(*
Nazwa:			GVL_VIS
Opis:			Zmienne dla wizualizacji
Wersja:			v0.2
Data:			2024-02-20
Autor:			MK
Urzadzenia:		
Konfiguracja:	
Info:
Zmiany:
- 20240220 [DP] Poprawki przed nowa wizką
*)

{attribute 'qualified_only'}
VAR_GLOBAL
	(*Legenda dla wizki :
		[H] - Hidden, prawdopodobnie nie potrzebne
		[I] - Info, informacja,
		[L] - Later, do zrobienia później, być może do przerobienia
	Uprawienia:
		brak opisu - operator
		[m] - Meechanik i powyżej
		[t] - Technolog i powyżej
		[s] - Serwis i powyżek
		[a] - Admin			
	*)

//-----------------------------------------CapSorterWheel--------------------------------------------------------------------------------------------------------------------------	
	//Sorter nasadek, koło
	iCapSorterWheelState							: INT;				// Stan
	sCapSorterWheelState							: STRING;   		// Stan
	bCapSorterWheelHoming							: BOOL;             // Bazowanie					// Przycisk bistabilny                     Bazowanie                                       									
	bCapSorterWheelManualWheelRight    				: BOOL;   			// Do przodu					// Przycisk monostabilny                     						
	bCapSorterWheelManualWheelLeft     				: BOOL;  			// Do tyłu						// Przycisk monostabilny  						
	bCapSorterWheelManualContinuousMovement			: BOOL;				// obrót o zadany kąt			// Przycisk bistabilny					
                                                                                               
//-----------------------------------------CapSorterCamera--------------------------------------------------------------------------------------------------------------------------	
	//Sorter nasadek, system wizyjny
	iCapSorterCameraState							: INT;				// Stan
	sCapSorterCameraState							: STRING;			// Stan
	bCapSorterCameraHoming							: BOOL;				// Bazowanie					// Przycisk bistabilny    	                                                	
	bCapSorterCameraManualRun						: BOOL;				// Zrób zdięcie					// Przycisk monostabilny
	bCapSorterBacklightManualStart					: BOOL;				// Podświetlenie stolu			// Przycisk bistabilny  
	uiCapSorterCameraActualJobIDLoaded				: UDINT;   	        // Program załadowany			// Pole do wyświetlania wartości                                   
	lrCapSorterCameraPickPointXVisu					: LREAL;			// Współrzędne produktu, X		// Pole do wyświetlania wartości
	lrCapSorterCameraPickPointYVisu					: LREAL;			// Współrzędne produktu, Y		// Pole do wyświetlania wartości
	lrCapSorterCameraPickPointAngleVisu				: LREAL;			// Kąt produktu					// Pole do wyświetlania wartości
                                                 	
//------------------------------------------ CapSorterRobot-------------------------------------------------------------------------------------------------------------------------	
	//Sorter nasadek, robot
	iCapSorterRobotState							: INT;				// Stan
	sCapSorterRobotState							: STRING;           // Stan
	bCapSorterRobotHoming							: BOOL;             // Bazowanie					// Przycisk bistabilny                                	
	
	bCapSorterRobotManualVacumOn					: BOOL; 			// Ssawka						// Przycisk bistabilny
	bCapSorterRobotManualRejectOn					: BOOL;				//Odrzut						// Przycisk bistabilny
	bCapSorterRobotManualGripperArmPosition1		: BOOL;  			// Ramię robota					// Przycisk bistabilny	
	bCapSorterRobotReadyPosition 					: BOOL;     		// Gotowość                                                                  	
	bCapSorterRobotPreparePick 						: BOOL;     		// Przygotuj do pobrania	
	bCapSorterRobotPick 							: BOOL;     		// Pobierz						// Przycisk bistabilny
	bCapSorterRobotPreparePlace						: BOOL;     		// Przygotuj do odłożenia
	bCapSorterRobotPlace							: BOOL;     		// Odłóż						// Przycisk bistabilny
	diCapSorterRobotPlaceId							: DINT; 			// Slot odłożenia | (1-4) 		// Pole do wpisywania wartosci
	diCapSorterRobotSpeed							: DINT; 			// Prędkość | [%] (1-100)		// Pole do wpisywania wartosci

		
//----------------------------------CapSorterTransporter---------------------------------------------------------------------------------------------------------------------------------
	//Sorter nasadek, transporter zasobnika
	iCapSorterTransporterState						: INT;				// Stan
	sCapSorterTransporterState						: STRING;           // Stan
	bCapSorterTransporterHoming						: BOOL;		        // Bazowanie					// Przycisk bistabilny                                          	
	bCapSorterTransporterManualTankConveyor			: BOOL;       		// Do przodu					// Przycisk bistabilny
	bCapSorterTransporterManualTankConveyorRevers	: BOOL;             // Do tyłu						// Przycisk bistabilny                                   	                                           	
		
	
	
//----------------------------------------CapSorterIntermediateTransporter---------------------------------------------------------------------------------------------------------------------------	
	// Sorter nasadek, transporter zasypowy
	iCapSorterIntermediateTransporterState			: INT;				// Stan
	sCapSorterIntermediateTransporterState			: STRING;	        // Stan                                      
	bCapSorterIntermediateTransporterHoming			: BOOL;             // Bazowanie					// Przycisk bistabilny   
	bCapSorterIntermediateTransporterManualForward	: BOOL;             // Do przodu					// Przycisk bistabilny
	bCapSorterIntermediateTransporterManualBackward	: BOOL;				// Do tyłu						// Przycisk bistabilny   
	
//----------------------------------------CapSorterIntermediateBrush---------------------------------------------------------------------------------------------------------------------------	
	//Sorter nasadek, szczotka transportera
	iCapSorterIntermediateBrushState				: INT;	  			// Stan
	sCapSorterIntermediateBrushState				: STRING;           // Stan
	bCapSorterIntermediateBrushHoming				: BOOL;             // Bazowanie					// Przycisk bistabilny                                      
	bCapSorterIntermediateBrushWeightSet			: BOOL;				// Ustaw pozycje				// Przycisk bistabilny
	bCapSorterIntermediateBrushManualForward		: BOOL;             // Do przodu					// Przycisk bistabilny
	bCapSorterIntermediateBrushManualBackward		: BOOL;		        // Do tyłu						// Przycisk bistabilny                                           
	bCapSorterIntermediateBrushManualLiftUp			: BOOL;				// Do góry						// Przycisk monostabilny
	bCapSorterIntermediateBrushManualLiftDown		: BOOL;             // Do dołu						// Przycisk monostabilny
	lrCapSorterIntermediateBrushActualHeight		: LREAL;			//Aktualna wysokosc | [mm]				// Pole do wyświetlania wartości
		
//-------------------------------------------CapSorterBrush1------------------------------------------------------------------------------------------------------------------------
	// Sorter nasadek, szczotka stolu 1
	iCapSorterBrush1OnWheelState					: INT;				// Stan
	sCapSorterBrush1OnWheelState					: STRING;           // Stan
	bCapSorterBrush1OnWheelHoming					: BOOL;	            // Bazowanie					// Przycisk bistabilny                                                       
	bCapSorterBrush1WeightSet						: BOOL;				// Ustaw pozycje				// Przycisk bistabilny
	bCapSorterBrush1OnWheelManualLiftUp				: BOOL;             // Do przodu					// Przycisk bistabilny
	bCapSorterBrush1OnWheelManualLiftDown			: BOOL;	            // Do tyłu						// Przycisk bistabilny                                                       
	bCapSorterBrush1OnWheelManualDriveForward		: BOOL;             // Do góry						// Przycisk monostabilny
	bCapSorterBrush1OnWheelManualDriveBackward		: BOOL;             // Do dołu						// Przycisk monostabilny
	lrCapSorterBrush1OnWheelActualHeight			: LREAL;	        //Aktualna wysokosc | [mm]				// Pole do wyświetlania wartości
	
//----------------------------------------CapSorterBrush2---------------------------------------------------------------------------------------------------------------------------	
	// Sorter nasadek, szczotka stolu 2
	iCapSorterBrush2State							: INT;				// Stan
	sCapSorterBrush2State							: STRING;           // Stan
	bCapSorterBrush2Homing							: BOOL;	            // Bazowanie					// Przycisk bistabilny                   
	bCapSorterBrush2WeightSet						: BOOL;				// Ustaw pozycje				// Przycisk bistabilny	
	bCapSorterBrushManualBrush2OnWheelLiftUp		: BOOL;             // Do przodu					// Przycisk bistabilny
	bCapSorterBrushManualBrush2OnWheelLiftDown		: BOOL;             // Do tyłu						// Przycisk bistabilny                   
	bCapSorterBrushManualBrush2OnWheelDriveForward	: BOOL;             // Do góry						// Przycisk monostabilny
	bCapSorterBrushManualBrush2OnWheelDriveBackward	: BOOL;             // Do dołu						// Przycisk monostabilny
	lrCapSorterBrush2OnWheelActualHeight			: LREAL;            //Aktualna wysokosc | [mm]				// Pole do wyświetlania wartości		

//-------------------------------------------------------------------------------------------------------------------------------------------------------------------	
	//Sorter nasadek, CapFeeder
	iCapSorterFeederState							: INT;			// Stan
	lrCapSorterFeederMover1CVShow					: LREAL;		// Pozycja mówera 1
	lrCapSorterFeederMover2CVShow					: LREAL;		// Pozycja mówera 2  
	sCapSorterFeederState							: STRING;       // Stan
	bCapSorterFeederHoming							: BOOL;			// Bazowanie						// Przycisk bistabilny 
	bCapSorterFeederMover1Forvard 					: BOOL;			// Mover 1 +						// Przycisk monostabilny
	bCapSorterFeederMover1Backward					: BOOL;			// Mover 1 -						// Przycisk monostabilny
	bCapSorterFeederMover2Forvard 					: BOOL;			// Mover 2 +						// Przycisk monostabilny
	bCapSorterFeederMover2Backward					: BOOL;			// Mover 2 -						// Przycisk monostabilny
	bCapSorterFeederMover1ActuatorIn				: BOOL;			// Mover 1 Do przodu				// Przycisk bistabilny
	bCapSorterFeederMover1ActuatorOut				: BOOL;			// Mover 1 Do tyłu					// Przycisk bistabilny
	bCapSorterFeederMover1PickPos					: BOOL;			// Mover 1, pozycja pobrania		// przycisk monostabilny
	bCapSorterFeederMover1PlacePos					: BOOL;			// Mover 1, pozycja odkładania		// przycisk monostabilny
	bCapSorterFeederMover2PickPos					: BOOL;			// Mover 2, pozycja pobrania		// przycisk monostabilny
	bCapSorterFeederMover2PlacePos					: BOOL;			// Mover 2, pozycja odkładania		// przycisk monostabilny
	
//-------------------------------------------------------------------------------------------------------------------------------------------------------------------	
	//Sorter nasadek, CapPreScrewer	
	iCapSorterPreScrewerState							: INT;			// Stan
	sCapSorterPreScrewerState							: STRING;       // Stan
	lrCapSorterPreScrewerYAxisCVShow					: LREAL;		// Pozycja kartezjana oś Y
	lrCapSorterPreScrewerZAxisCVShow					: LREAL;		// Pozycja kartezjana oś Z
	lrCapSorterPreScrewerCAxisCVShow					: LREAL;		// Pozycja kartezjana oś C  
	bCapSorterPreScrewerHoming							: BOOL;			// Bazowanie					// Przycisk bistabilny 
	bCapSorterPreScrewerSetOffsetEncoderAxisZ			: BOOL;			// Ustaw offset encodera osi Z	//	Przycisk monostabilny
	bCapSorterPreScrewerPicker1Catch					: BOOL;			// Chwytak 1					// 	Przycisk bistabilny 
	bCapSorterPreScrewerPicker2Catch					: BOOL;			// Chwytak 2					// 	Przycisk bistabilny 
	bCapSorterPreScrewerPicker3Catch					: BOOL;			// Chwytak 3					// 	Przycisk bistabilny 
	bCapSorterPreScrewerPicker4Catch					: BOOL;			// Chwytak 4					// 	Przycisk bistabilny 
	bCapSorterPreScrewerPicker1Vacuum					: BOOL;			// Podsys 1						// 	Przycisk bistabilny 	
	bCapSorterPreScrewerPicker2Vacuum					: BOOL;			// Podsys 2						// 	Przycisk bistabilny 	
	bCapSorterPreScrewerPicker3Vacuum					: BOOL;			// Podsys 3						// 	Przycisk bistabilny 	
	bCapSorterPreScrewerPicker4Vacuum					: BOOL;			// Podsys 4						// 	Przycisk bistabilny 	
	bCapSorterPreScrewerPicker1Reject					: BOOL;			// Oddmuch 1					// 	Przycisk bistabilny	
	bCapSorterPreScrewerPicker2Reject					: BOOL;			// Oddmuch 2					// 	Przycisk bistabilny	
	bCapSorterPreScrewerPicker3Reject					: BOOL;			// Oddmuch 3					// 	Przycisk bistabilny	
	bCapSorterPreScrewerPicker4Reject					: BOOL;			// Oddmuch 4					// 	Przycisk bistabilny	
	
		//Kartezjan
	bCapSorterPreScrewerCartesianYForward				: BOOL;			// Y +							// Przycisk monostabilny
	bCapSorterPreScrewerCartesianYBackward				: BOOL;			// Y -							// Przycisk monostabilny
	bCapSorterPreScrewerCartesianZForward				: BOOL;			// Z +							// Przycisk monostabilny
	bCapSorterPreScrewerCartesianZBackward				: BOOL;			// Z -							// Przycisk monostabilny
	bCapSorterPreScrewerCartesianCForward				: BOOL;			// C +							// Przycisk monostabilny
	bCapSorterPreScrewerCartesianCBackward				: BOOL;			// C -							// Przycisk monostabilny
	                                                    	        	
		//Łapacz słomki    
 	lrCapSorterPreScrewerStrawCatcherCVShow				: LREAL;		// Pozycja łapacza słomek                           	
    bCapSorterPreScrewerStrawCatcherUp					: BOOL;			// Chwytaki do góry 			// Przycisk monostabilny
	bCapSorterPreScrewerStrawCatcherDown				: BOOL;			// Chwytaki do dołu 			// Przycisk monostabilny	
	bCapSorterPreScrewerStrawCatcherCatchOpen			: BOOL;			// Otwórz chwytaki słomek		// Przycisk bistabilny
	bCapSorterPreScrewerStrawCatcherCatchClose			: BOOL;			// Zamknij chwytaki słomek		// Przycisk bistabilny
	bCapSorterPreScrewerStrawCatcherActuatorIn			: BOOL;			//  Wsuń łapacz słomek			// Przycisk bistabilny
	bCapSorterPreScrewerStrawCatcherActuatorOut			: BOOL;			//  Wysuń łapacz słomek			// Przycisk bistabilny
                                                    	

                                                		
		//Podnośnik stacji wkladania nakrętek       		            	 
	bCapSorterPreScrewerCatcherStationUp					: BOOL;			// Stacja do góry 				// Przycisk monostabilny
	bCapSorterPreScrewerCatcherStationDown					: BOOL;			// Stacja do dołu 				// Przycisk monostabilny                 			
	bCapSorterPreScrewerBottleCatcherCatch					: BOOL;			// Chwytaki Butelek				// Przycisk bistabilny	
	lrCapSorterPreScrewerCatcherStationHeightCV				: LREAL;		// Aktualna wysokość chwytaka
	bCapSorterPreScrewerCatcherStationHeightSet				: BOOL;			// Ustaw pozycje				// Przycisk bistabilny
	bCapSorterPreScrewerBottleCatchOpenCalibration			: BOOL;			// Kalibruj otwarcie			// Przycisk bistabilny
	bCapSorterPreScrewerBottleCatchCloseCalibration			: BOOL;			// Kalibruj zamknięcie			// Przycisk bistabilny
	bCapSorterPreScrewerNextStep							: BOOL;			// Kolejny krok w serwice mode
                                                                        
	//Chwytak szyjki butelki pod wkladaczem nakrentek 1234                  
	bCapSorterPreScrewerCatchStationHoming	      			: BOOL;			// [H] Homing  					// Przycisk bistabilny	
	lrCapSorterPreScrewerCatchStationHeightSVShow			: LREAL;  		// Pozycja chwytaka
	bCapSorterPreScrewerManualBottleCatcherCatch			: BOOL;											// Przycisk bistabilny	        
 	
	
	bCapSorterManualVacuumPump								: BOOL; 
	// 1-Fliptop (prosta scieżka), 2-Pompka/Atomizer (Stawianie do pionu), 3-Fliptop z boku (stawianie do pionu + detekcja obróconej)
	AsCapSorterProductType									: ARRAY [1..10] OF STRING;
//	iCapSorterProductType									: INT;
	//
	AsCapSorterIndexShow									: ARRAY [1..30] OF STRING;	
//	uiCapSorterIndexShow									: UDINT;
	

	bCapSorterFeederAdvancedHoming							: BOOL;			// Bazowanie wózków "na zderzak"	
	bCapSorterPreScrewerAdvancedHoming						: BOOL;			// Bazowanie zaawansowane dotyczy osi Y
	
	lrCapSorterPreScrewerVacuumLevel_1						: LREAL;			// Podcisnienie na głowicy nr1	[Bar]
	lrCapSorterPreScrewerVacuumLevel_2						: LREAL;			// Podcisnienie na głowicy nr2	[Bar]
	lrCapSorterPreScrewerVacuumLevel_3						: LREAL;			// Podcisnienie na głowicy nr3	[Bar]
	lrCapSorterPreScrewerVacuumLevel_4						: LREAL;			// Podcisnienie na głowicy nr4	[Bar]	
	
//-----------------------------------------------------------------------------------------------------------------------------------------------------

	bCapSorterCalculateParameters							: BOOL;			//	Oblicz paramaretry maszyny	//przycisk monostabilny
	bCapSorterSpare1										: BOOL;			//Rezerwa 1
	bCapSorterSpare2										: BOOL;			//Rezerwa 2
	bCapSorterSpare3										: BOOL;			//Rezerwa 3
	bCapSorterSpare4										: BOOL;			//Rezerwa 4
	bCapSorterSpare5										: BOOL;			//Rezerwa 5
	bCapSorterSpare6										: BOOL;			//Rezerwa 6
	bCapSorterSpare7										: BOOL;			//Rezerwa 7
	
	fbAlarms :FB_Events; 	//ActiveAlarms
	
	
END_VAR

(* stored: Version 1.2.0.0, ProductVersion 3.1.4026.13, FileIdentifier 39b673a7309509a6b0fd60dd2def5df56f797a54, FileSignature 939292e2fd8c47996c99e1d1c56bd5e012c541e44475e5a4f0c9c5999af3d1650c5f531b261fa3c2bd795daab5ede88473159e4182be54dc6d57dd99411602f353faf693430527fa29613c16a411e01f410016fd914910b5411664334905648b6df06498c55b8218a1780f6d7a5f77c44d27c350c417b8e055cbf94bd37e33a925a1e11a8c2a01cfd26530400008ae4203d6b77e0ee06e158ebc207b2d53c77c50e70f1c6e080953212f8aad0b374ddb7371d031a38dd9a2f82924dde79d76d67eeae62d23815216dcdd314da8730bd271e1fd5992cdbc752006b7f49bf023ab7b4911849061a7a603da4cb6d25f5bccf16c5a8b27d675f4e1b4e13125d8b969
   GVL GVL_VIS: Id {0555371b-99ed-4592-8d57-d012452c0e38} *)
